// TIA Portal V20 export
TYPE "LER_TypeFATMode_Sampling_SetValue"
// stored: Access Published
   STRUCT
      SelectCount_SetValue : Int;
   END_STRUCT;
END_TYPE
